PROGRAM MAIN
VAR
	fbErrorHandler: FB_ErrorHandler;
	fbBoiler1: FB_Boiler;
	fbBoiler2: FB_Boiler;
END_VAR


fbBoiler1(itfErrorHandler:=fbErrorHandler );
fbBoiler2(itfErrorHandler:=fbErrorHandler );

fbErrorHandler();

END_PROGRAM

(* stored: Version 1.1.0.1, ProductVersion 3.1.4024.11
   POU MAIN: Id {cbe91a83-74aa-4d62-b058-d6d2b5d624db}, SpecialFunc None *)
